INTERFACE ITF_GroupElement_HMI_Init EXTENDS ITF_BaseGroupElement, ITF_GroupElement_HMI_Connector

END_INTERFACE

(* stored: Version 1.1.0.1, ProductVersion 3.1.4024.15
   Itf ITF_GroupElement_HMI_Init: Id {310885a6-d417-426c-80b6-5120d1ea6710} *)
